TYPE ST_ManualModeKeyHWUnit :
STRUCT
	nLogAxisId: UINT;
	nChan: INT := -1;
	nInputParameterIdx: INT;
END_STRUCT
END_TYPE

(* stored: Version 1.1.0.1, ProductVersion 3.1.4019.0
   DUT ST_ManualModeKeyHWUnit: Id {34218d39-97f3-450d-9ca3-73082542f3ab} *)
